// Mitsubishi GX Works2 project: k11   PLC: Q02/Q02H

PROGRAM MAIN
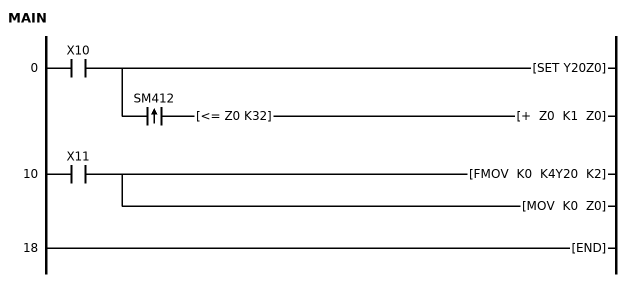
0     LD      X10
      SET     Y20Z0
      ANDP    SM412
      AND<=   Z0 K32
      +       Z0 K1 Z0
10    LD      X11
      FMOV    K0 K4Y20 K2
      MOV     K0 Z0
18    END
END_PROGRAM
